Fanuc KAREL source: kb00107.KL

PROGRAM KB00107
%STACKSIZE=65535
%PRIORITY=65535
%NOLOCKGROUP
VAR
P1 : XYZWPREXT
RESULT : BOOLEAN
BEGIN
-- UNRESOLVED_PC line 7 opcodes [27 22 1C 27 9D 76 23] marker_code=0
END KB00107
